// Mitsubishi GX Works2 project: HMI 연습용 PLC 코드   PLC: Q03UDV

PROGRAM MAIN
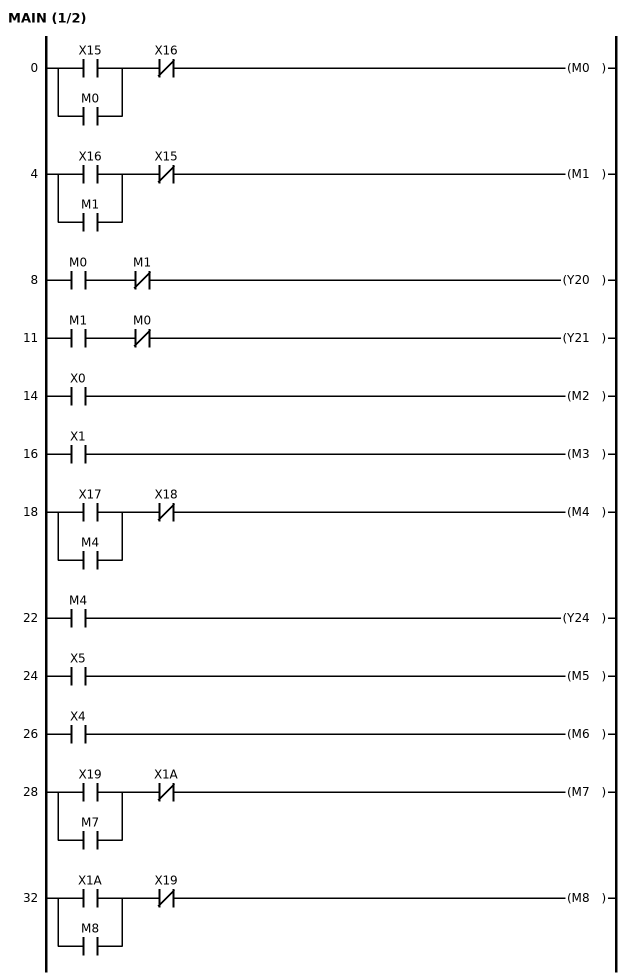
0     LD      X15
      OR      M0
      ANI     X16
      OUT     M0
4     LD      X16
      OR      M1
      ANI     X15
      OUT     M1
8     LD      M0
      ANI     M1
      OUT     Y20
11    LD      M1
      ANI     M0
      OUT     Y21
14    LD      X0
      OUT     M2
16    LD      X1
      OUT     M3
18    LD      X17
      OR      M4
      ANI     X18
      OUT     M4
22    LD      M4
      OUT     Y24
24    LD      X5
      OUT     M5
26    LD      X4
      OUT     M6
28    LD      X19
      OR      M7
      ANI     X1A
      OUT     M7
32    LD      X1A
      OR      M8
      ANI     X19
      OUT     M8
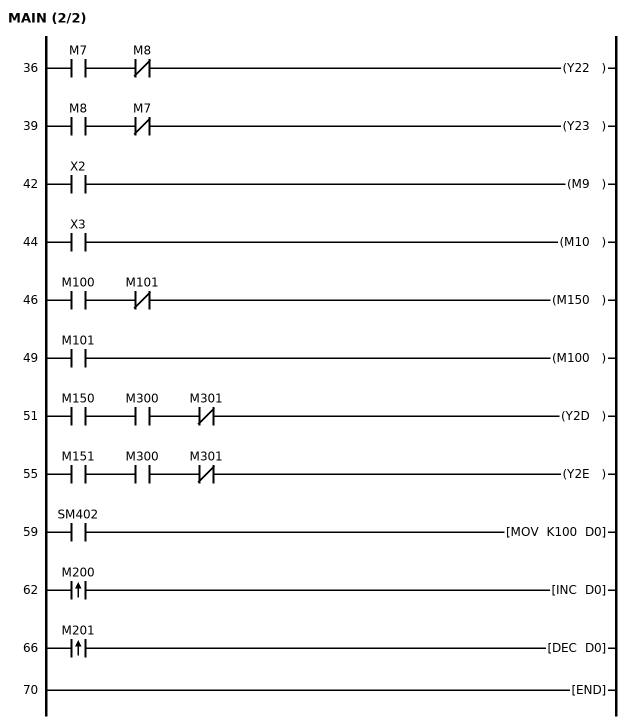
36    LD      M7
      ANI     M8
      OUT     Y22
39    LD      M8
      ANI     M7
      OUT     Y23
42    LD      X2
      OUT     M9
44    LD      X3
      OUT     M10
46    LD      M100
      ANI     M101
      OUT     M150
49    LD      M101
      OUT     M100
51    LD      M150
      AND     M300
      ANI     M301
      OUT     Y2D
55    LD      M151
      AND     M300
      ANI     M301
      OUT     Y2E
59    LD      SM402
      MOV     K100 D0
62    LDP     M200
      INC     D0
66    LDP     M201
      DEC     D0
70    END
END_PROGRAM
